(* IEC 61131-3 sources: Simulated-machine/integrations/openplc/thermal-plant-v3, 1 file *)

(* ---- thermal-plant-v3.st ---- *)
(* Generated by tools/generate_openplc_v3_gateway.py.
   OpenPLC Runtime v3 gateway for the self-holding thermal plant.

   The devices start themselves and run their own regulators.  This
   program only exchanges data and evaluates logic; it never computes a
   control value.  The only holding registers written are
   COMMAND_SEQUENCE, WATCHDOG_COUNTER and RESET_KEY.

   Addresses come from the OpenPLC v3 Modbus master image: slave devices
   must be configured in the order listed in slave-devices.csv. *)
PROGRAM main
  VAR
    i_outputs_initialized : BOOL := FALSE;
    i_watchdog_scan_count : UINT := 0;
    i_watchdog_tick : BOOL := FALSE;
    i_plant_comm_lost : BOOL := FALSE;
    i_overspeed : BOOL := FALSE;
    i_overspeed_prev : BOOL := FALSE;
    i_condenser_last_echo : UINT := 0;
    i_condenser_echo_stale_ticks : UINT := 0;
    i_condenser_comm_lost : BOOL := FALSE;
    i_condensate_pump_last_echo : UINT := 0;
    i_condensate_pump_echo_stale_ticks : UINT := 0;
    i_condensate_pump_comm_lost : BOOL := FALSE;
    i_feedwater_tank_last_echo : UINT := 0;
    i_feedwater_tank_echo_stale_ticks : UINT := 0;
    i_feedwater_tank_comm_lost : BOOL := FALSE;
    i_feedwater_pump_last_echo : UINT := 0;
    i_feedwater_pump_echo_stale_ticks : UINT := 0;
    i_feedwater_pump_comm_lost : BOOL := FALSE;
    i_boiler_last_echo : UINT := 0;
    i_boiler_echo_stale_ticks : UINT := 0;
    i_boiler_comm_lost : BOOL := FALSE;
    i_steam_valve_last_echo : UINT := 0;
    i_steam_valve_echo_stale_ticks : UINT := 0;
    i_steam_valve_comm_lost : BOOL := FALSE;
    i_turbine_last_echo : UINT := 0;
    i_turbine_echo_stale_ticks : UINT := 0;
    i_turbine_comm_lost : BOOL := FALSE;
    i_generator_last_echo : UINT := 0;
    i_generator_echo_stale_ticks : UINT := 0;
    i_generator_comm_lost : BOOL := FALSE;
    i_condenser_start_active : BOOL := FALSE;
    i_condenser_start_scans : UINT := 0;
    i_condenser_stop_active : BOOL := FALSE;
    i_condenser_stop_scans : UINT := 0;
    i_condenser_reset_trip_active : BOOL := FALSE;
    i_condenser_reset_trip_scans : UINT := 0;
    i_condenser_ack_alarm_active : BOOL := FALSE;
    i_condenser_ack_alarm_scans : UINT := 0;
    i_condenser_trip_test_active : BOOL := FALSE;
    i_condenser_trip_test_scans : UINT := 0;
    i_condenser_clear_totalizer_active : BOOL := FALSE;
    i_condenser_clear_totalizer_scans : UINT := 0;
    i_condensate_pump_start_active : BOOL := FALSE;
    i_condensate_pump_start_scans : UINT := 0;
    i_condensate_pump_stop_active : BOOL := FALSE;
    i_condensate_pump_stop_scans : UINT := 0;
    i_condensate_pump_reset_trip_active : BOOL := FALSE;
    i_condensate_pump_reset_trip_scans : UINT := 0;
    i_condensate_pump_ack_alarm_active : BOOL := FALSE;
    i_condensate_pump_ack_alarm_scans : UINT := 0;
    i_condensate_pump_trip_test_active : BOOL := FALSE;
    i_condensate_pump_trip_test_scans : UINT := 0;
    i_condensate_pump_clear_totalizer_active : BOOL := FALSE;
    i_condensate_pump_clear_totalizer_scans : UINT := 0;
    i_feedwater_tank_start_active : BOOL := FALSE;
    i_feedwater_tank_start_scans : UINT := 0;
    i_feedwater_tank_stop_active : BOOL := FALSE;
    i_feedwater_tank_stop_scans : UINT := 0;
    i_feedwater_tank_reset_trip_active : BOOL := FALSE;
    i_feedwater_tank_reset_trip_scans : UINT := 0;
    i_feedwater_tank_ack_alarm_active : BOOL := FALSE;
    i_feedwater_tank_ack_alarm_scans : UINT := 0;
    i_feedwater_tank_trip_test_active : BOOL := FALSE;
    i_feedwater_tank_trip_test_scans : UINT := 0;
    i_feedwater_tank_clear_totalizer_active : BOOL := FALSE;
    i_feedwater_tank_clear_totalizer_scans : UINT := 0;
    i_feedwater_pump_start_active : BOOL := FALSE;
    i_feedwater_pump_start_scans : UINT := 0;
    i_feedwater_pump_stop_active : BOOL := FALSE;
    i_feedwater_pump_stop_scans : UINT := 0;
    i_feedwater_pump_reset_trip_active : BOOL := FALSE;
    i_feedwater_pump_reset_trip_scans : UINT := 0;
    i_feedwater_pump_ack_alarm_active : BOOL := FALSE;
    i_feedwater_pump_ack_alarm_scans : UINT := 0;
    i_feedwater_pump_trip_test_active : BOOL := FALSE;
    i_feedwater_pump_trip_test_scans : UINT := 0;
    i_feedwater_pump_clear_totalizer_active : BOOL := FALSE;
    i_feedwater_pump_clear_totalizer_scans : UINT := 0;
    i_boiler_start_active : BOOL := FALSE;
    i_boiler_start_scans : UINT := 0;
    i_boiler_stop_active : BOOL := FALSE;
    i_boiler_stop_scans : UINT := 0;
    i_boiler_reset_trip_active : BOOL := FALSE;
    i_boiler_reset_trip_scans : UINT := 0;
    i_boiler_ack_alarm_active : BOOL := FALSE;
    i_boiler_ack_alarm_scans : UINT := 0;
    i_boiler_trip_test_active : BOOL := FALSE;
    i_boiler_trip_test_scans : UINT := 0;
    i_boiler_clear_totalizer_active : BOOL := FALSE;
    i_boiler_clear_totalizer_scans : UINT := 0;
    i_steam_valve_start_active : BOOL := FALSE;
    i_steam_valve_start_scans : UINT := 0;
    i_steam_valve_stop_active : BOOL := FALSE;
    i_steam_valve_stop_scans : UINT := 0;
    i_steam_valve_reset_trip_active : BOOL := FALSE;
    i_steam_valve_reset_trip_scans : UINT := 0;
    i_steam_valve_ack_alarm_active : BOOL := FALSE;
    i_steam_valve_ack_alarm_scans : UINT := 0;
    i_steam_valve_trip_test_active : BOOL := FALSE;
    i_steam_valve_trip_test_scans : UINT := 0;
    i_steam_valve_clear_totalizer_active : BOOL := FALSE;
    i_steam_valve_clear_totalizer_scans : UINT := 0;
    i_turbine_start_active : BOOL := FALSE;
    i_turbine_start_scans : UINT := 0;
    i_turbine_stop_active : BOOL := FALSE;
    i_turbine_stop_scans : UINT := 0;
    i_turbine_reset_trip_active : BOOL := FALSE;
    i_turbine_reset_trip_scans : UINT := 0;
    i_turbine_ack_alarm_active : BOOL := FALSE;
    i_turbine_ack_alarm_scans : UINT := 0;
    i_turbine_trip_test_active : BOOL := FALSE;
    i_turbine_trip_test_scans : UINT := 0;
    i_turbine_clear_totalizer_active : BOOL := FALSE;
    i_turbine_clear_totalizer_scans : UINT := 0;
    i_generator_start_active : BOOL := FALSE;
    i_generator_start_scans : UINT := 0;
    i_generator_stop_active : BOOL := FALSE;
    i_generator_stop_scans : UINT := 0;
    i_generator_reset_trip_active : BOOL := FALSE;
    i_generator_reset_trip_scans : UINT := 0;
    i_generator_ack_alarm_active : BOOL := FALSE;
    i_generator_ack_alarm_scans : UINT := 0;
    i_generator_trip_test_active : BOOL := FALSE;
    i_generator_trip_test_scans : UINT := 0;
    i_generator_clear_totalizer_active : BOOL := FALSE;
    i_generator_clear_totalizer_scans : UINT := 0;
    i_turbine_trip_prev : BOOL := FALSE;
    i_boiler_trip_prev : BOOL := FALSE;
    i_condenser_trip_prev : BOOL := FALSE;
    i_feedwater_pump_trip_prev : BOOL := FALSE;
    i_condensate_pump_trip_prev : BOOL := FALSE;
    i_steam_valve_trip_prev : BOOL := FALSE;

    condenser__coil__start AT %QX100.0 : BOOL := FALSE;
    condenser__coil__stop AT %QX100.1 : BOOL := FALSE;
    condenser__coil__reset_trip AT %QX100.2 : BOOL := FALSE;
    condenser__coil__ack_alarm AT %QX100.3 : BOOL := FALSE;
    condenser__coil__emergency_stop AT %QX100.4 : BOOL := FALSE;
    condenser__coil__force_safe AT %QX100.5 : BOOL := FALSE;
    condenser__coil__trip_test AT %QX100.6 : BOOL := FALSE;
    condenser__coil__clear_totalizer AT %QX100.7 : BOOL := FALSE;
    condenser__discrete__ready AT %IX100.0 : BOOL := FALSE;
    condenser__discrete__running AT %IX100.1 : BOOL := FALSE;
    condenser__discrete__starting AT %IX100.2 : BOOL := FALSE;
    condenser__discrete__stopping AT %IX100.3 : BOOL := FALSE;
    condenser__discrete__tripped AT %IX100.4 : BOOL := FALSE;
    condenser__discrete__alarm_active AT %IX100.5 : BOOL := FALSE;
    condenser__discrete__local_mode AT %IX100.6 : BOOL := FALSE;
    condenser__discrete__remote_mode AT %IX100.7 : BOOL := FALSE;
    condenser__discrete__auto_mode AT %IX101.0 : BOOL := FALSE;
    condenser__discrete__manual_mode AT %IX101.1 : BOOL := FALSE;
    condenser__discrete__control_watchdog_ok AT %IX101.2 : BOOL := FALSE;
    condenser__discrete__sim_bus_ok AT %IX101.3 : BOOL := FALSE;
    condenser__discrete__interlocks_ok AT %IX101.4 : BOOL := FALSE;
    condenser__discrete__sensor_fault AT %IX101.5 : BOOL := FALSE;
    condenser__discrete__actuator_fault AT %IX101.6 : BOOL := FALSE;
    condenser__discrete__maintenance_mode AT %IX101.7 : BOOL := FALSE;
    condenser__input__status_word AT %IW100 : UINT := 0;
    condenser__input__alarm_word_1 AT %IW101 : UINT := 0;
    condenser__input__alarm_word_2 AT %IW102 : UINT := 0;
    condenser__input__trip_word AT %IW103 : UINT := 0;
    condenser__input__device_state AT %IW104 : UINT := 0;
    condenser__input__first_out_code AT %IW105 : UINT := 0;
    condenser__input__overall_quality AT %IW106 : UINT := 0;
    condenser__input__register_map_version AT %IW107 : UINT := 0;
    condenser__input__firmware_version AT %IW108 : UINT := 0;
    condenser__input__condenser_pressure AT %IW109 : UINT := 0;
    condenser__input__vacuum AT %IW110 : UINT := 0;
    condenser__input__hotwell_level AT %IW111 : UINT := 0;
    condenser__input__exhaust_inflow AT %IW112 : UINT := 0;
    condenser__input__condensing_capacity AT %IW113 : UINT := 0;
    condenser__input__actual_condensed AT %IW114 : UINT := 0;
    condenser__input__condensate_outflow AT %IW115 : UINT := 0;
    condenser__input__cooling_water_availability AT %IW116 : UINT := 0;
    condenser__input__vacuum_system_output AT %IW117 : UINT := 0;
    condenser__input__condensate_temperature AT %IW118 : UINT := 0;
    condenser__input__hotwell_mass_hi AT %IW119 : UINT := 0;
    condenser__input__hotwell_mass_lo AT %IW120 : UINT := 0;
    condenser__input__makeup_valve_position AT %IW121 : UINT := 0;
    condenser__input__makeup_flow AT %IW122 : UINT := 0;
    condenser__input__local_output AT %IW125 : UINT := 0;
    condenser__input__self_hold_state AT %IW126 : UINT := 0;
    condenser__input__permissive_word AT %IW127 : UINT := 0;
    condenser__input__watchdog_echo AT %IW129 : UINT := 0;
    condenser__input__scan_time_ms AT %IW130 : UINT := 0;
    condenser__input__modbus_request_count AT %IW131 : UINT := 0;
    condenser__input__rejected_command_count AT %IW132 : UINT := 0;
    condenser__input__exception_count AT %IW133 : UINT := 0;
    condenser__input__sim_quality_word AT %IW134 : UINT := 0;
    condenser__input__sim_tick_low AT %IW135 : UINT := 0;
    condenser__input__comm_loss_seconds AT %IW136 : UINT := 0;
    condenser__input__fault_inject_word AT %IW137 : UINT := 0;
    condenser__input__snapshot_generation AT %IW138 : UINT := 0;
    condenser__input__run_seconds_hi AT %IW139 : UINT := 0;
    condenser__input__run_seconds_lo AT %IW140 : UINT := 0;
    condenser__input__start_count AT %IW141 : UINT := 0;
    condenser__input__trip_count AT %IW142 : UINT := 0;
    condenser__input__mass_total_hi AT %IW143 : UINT := 0;
    condenser__input__mass_total_lo AT %IW144 : UINT := 0;
    condenser__input__energy_total_hi AT %IW145 : UINT := 0;
    condenser__input__energy_total_lo AT %IW146 : UINT := 0;
    condenser__input__alarm_count AT %IW147 : UINT := 0;
    condenser__input__accepted_command_count AT %IW148 : UINT := 0;
    condenser__holding__command_sequence AT %QW100 : UINT := 0;
    condenser__holding__watchdog_counter AT %QW101 : UINT := 0;
    condenser__holding__reset_key AT %QW102 : UINT := 0;
    condensate_pump__coil__start AT %QX101.0 : BOOL := FALSE;
    condensate_pump__coil__stop AT %QX101.1 : BOOL := FALSE;
    condensate_pump__coil__reset_trip AT %QX101.2 : BOOL := FALSE;
    condensate_pump__coil__ack_alarm AT %QX101.3 : BOOL := FALSE;
    condensate_pump__coil__emergency_stop AT %QX101.4 : BOOL := FALSE;
    condensate_pump__coil__force_safe AT %QX101.5 : BOOL := FALSE;
    condensate_pump__coil__trip_test AT %QX101.6 : BOOL := FALSE;
    condensate_pump__coil__clear_totalizer AT %QX101.7 : BOOL := FALSE;
    condensate_pump__discrete__ready AT %IX102.0 : BOOL := FALSE;
    condensate_pump__discrete__running AT %IX102.1 : BOOL := FALSE;
    condensate_pump__discrete__starting AT %IX102.2 : BOOL := FALSE;
    condensate_pump__discrete__stopping AT %IX102.3 : BOOL := FALSE;
    condensate_pump__discrete__tripped AT %IX102.4 : BOOL := FALSE;
    condensate_pump__discrete__alarm_active AT %IX102.5 : BOOL := FALSE;
    condensate_pump__discrete__local_mode AT %IX102.6 : BOOL := FALSE;
    condensate_pump__discrete__remote_mode AT %IX102.7 : BOOL := FALSE;
    condensate_pump__discrete__auto_mode AT %IX103.0 : BOOL := FALSE;
    condensate_pump__discrete__manual_mode AT %IX103.1 : BOOL := FALSE;
    condensate_pump__discrete__control_watchdog_ok AT %IX103.2 : BOOL := FALSE;
    condensate_pump__discrete__sim_bus_ok AT %IX103.3 : BOOL := FALSE;
    condensate_pump__discrete__interlocks_ok AT %IX103.4 : BOOL := FALSE;
    condensate_pump__discrete__sensor_fault AT %IX103.5 : BOOL := FALSE;
    condensate_pump__discrete__actuator_fault AT %IX103.6 : BOOL := FALSE;
    condensate_pump__discrete__maintenance_mode AT %IX103.7 : BOOL := FALSE;
    condensate_pump__input__status_word AT %IW149 : UINT := 0;
    condensate_pump__input__alarm_word_1 AT %IW150 : UINT := 0;
    condensate_pump__input__alarm_word_2 AT %IW151 : UINT := 0;
    condensate_pump__input__trip_word AT %IW152 : UINT := 0;
    condensate_pump__input__device_state AT %IW153 : UINT := 0;
    condensate_pump__input__first_out_code AT %IW154 : UINT := 0;
    condensate_pump__input__overall_quality AT %IW155 : UINT := 0;
    condensate_pump__input__register_map_version AT %IW156 : UINT := 0;
    condensate_pump__input__firmware_version AT %IW157 : UINT := 0;
    condensate_pump__input__actual_speed AT %IW158 : UINT := 0;
    condensate_pump__input__flow AT %IW159 : UINT := 0;
    condensate_pump__input__suction_pressure AT %IW160 : UINT := 0;
    condensate_pump__input__discharge_pressure AT %IW161 : UINT := 0;
    condensate_pump__input__motor_current AT %IW162 : UINT := 0;
    condensate_pump__input__npsh_margin AT %IW163 : UINT := 0;
    condensate_pump__input__vibration AT %IW164 : UINT := 0;
    condensate_pump__input__source_level AT %IW165 : UINT := 0;
    condensate_pump__input__backpressure AT %IW166 : UINT := 0;
    condensate_pump__input__outlet_valve_position AT %IW167 : UINT := 0;
    condensate_pump__input__cavitation_factor AT %IW168 : UINT := 0;
    condensate_pump__input__local_output AT %IW174 : UINT := 0;
    condensate_pump__input__self_hold_state AT %IW175 : UINT := 0;
    condensate_pump__input__permissive_word AT %IW176 : UINT := 0;
    condensate_pump__input__watchdog_echo AT %IW178 : UINT := 0;
    condensate_pump__input__scan_time_ms AT %IW179 : UINT := 0;
    condensate_pump__input__modbus_request_count AT %IW180 : UINT := 0;
    condensate_pump__input__rejected_command_count AT %IW181 : UINT := 0;
    condensate_pump__input__exception_count AT %IW182 : UINT := 0;
    condensate_pump__input__sim_quality_word AT %IW183 : UINT := 0;
    condensate_pump__input__sim_tick_low AT %IW184 : UINT := 0;
    condensate_pump__input__comm_loss_seconds AT %IW185 : UINT := 0;
    condensate_pump__input__fault_inject_word AT %IW186 : UINT := 0;
    condensate_pump__input__snapshot_generation AT %IW187 : UINT := 0;
    condensate_pump__input__run_seconds_hi AT %IW188 : UINT := 0;
    condensate_pump__input__run_seconds_lo AT %IW189 : UINT := 0;
    condensate_pump__input__start_count AT %IW190 : UINT := 0;
    condensate_pump__input__trip_count AT %IW191 : UINT := 0;
    condensate_pump__input__mass_total_hi AT %IW192 : UINT := 0;
    condensate_pump__input__mass_total_lo AT %IW193 : UINT := 0;
    condensate_pump__input__energy_total_hi AT %IW194 : UINT := 0;
    condensate_pump__input__energy_total_lo AT %IW195 : UINT := 0;
    condensate_pump__input__alarm_count AT %IW196 : UINT := 0;
    condensate_pump__input__accepted_command_count AT %IW197 : UINT := 0;
    condensate_pump__holding__command_sequence AT %QW103 : UINT := 0;
    condensate_pump__holding__watchdog_counter AT %QW104 : UINT := 0;
    condensate_pump__holding__reset_key AT %QW105 : UINT := 0;
    feedwater_tank__coil__start AT %QX102.0 : BOOL := FALSE;
    feedwater_tank__coil__stop AT %QX102.1 : BOOL := FALSE;
    feedwater_tank__coil__reset_trip AT %QX102.2 : BOOL := FALSE;
    feedwater_tank__coil__ack_alarm AT %QX102.3 : BOOL := FALSE;
    feedwater_tank__coil__emergency_stop AT %QX102.4 : BOOL := FALSE;
    feedwater_tank__coil__force_safe AT %QX102.5 : BOOL := FALSE;
    feedwater_tank__coil__trip_test AT %QX102.6 : BOOL := FALSE;
    feedwater_tank__coil__clear_totalizer AT %QX102.7 : BOOL := FALSE;
    feedwater_tank__discrete__ready AT %IX104.0 : BOOL := FALSE;
    feedwater_tank__discrete__running AT %IX104.1 : BOOL := FALSE;
    feedwater_tank__discrete__starting AT %IX104.2 : BOOL := FALSE;
    feedwater_tank__discrete__stopping AT %IX104.3 : BOOL := FALSE;
    feedwater_tank__discrete__tripped AT %IX104.4 : BOOL := FALSE;
    feedwater_tank__discrete__alarm_active AT %IX104.5 : BOOL := FALSE;
    feedwater_tank__discrete__local_mode AT %IX104.6 : BOOL := FALSE;
    feedwater_tank__discrete__remote_mode AT %IX104.7 : BOOL := FALSE;
    feedwater_tank__discrete__auto_mode AT %IX105.0 : BOOL := FALSE;
    feedwater_tank__discrete__manual_mode AT %IX105.1 : BOOL := FALSE;
    feedwater_tank__discrete__control_watchdog_ok AT %IX105.2 : BOOL := FALSE;
    feedwater_tank__discrete__sim_bus_ok AT %IX105.3 : BOOL := FALSE;
    feedwater_tank__discrete__interlocks_ok AT %IX105.4 : BOOL := FALSE;
    feedwater_tank__discrete__sensor_fault AT %IX105.5 : BOOL := FALSE;
    feedwater_tank__discrete__actuator_fault AT %IX105.6 : BOOL := FALSE;
    feedwater_tank__discrete__maintenance_mode AT %IX105.7 : BOOL := FALSE;
    feedwater_tank__input__status_word AT %IW198 : UINT := 0;
    feedwater_tank__input__alarm_word_1 AT %IW199 : UINT := 0;
    feedwater_tank__input__alarm_word_2 AT %IW200 : UINT := 0;
    feedwater_tank__input__trip_word AT %IW201 : UINT := 0;
    feedwater_tank__input__device_state AT %IW202 : UINT := 0;
    feedwater_tank__input__first_out_code AT %IW203 : UINT := 0;
    feedwater_tank__input__overall_quality AT %IW204 : UINT := 0;
    feedwater_tank__input__register_map_version AT %IW205 : UINT := 0;
    feedwater_tank__input__firmware_version AT %IW206 : UINT := 0;
    feedwater_tank__input__tank_level AT %IW207 : UINT := 0;
    feedwater_tank__input__tank_mass_hi AT %IW208 : UINT := 0;
    feedwater_tank__input__tank_mass_lo AT %IW209 : UINT := 0;
    feedwater_tank__input__condensate_inflow AT %IW210 : UINT := 0;
    feedwater_tank__input__feedwater_outflow AT %IW211 : UINT := 0;
    feedwater_tank__input__water_temperature AT %IW212 : UINT := 0;
    feedwater_tank__input__tank_pressure AT %IW213 : UINT := 0;
    feedwater_tank__input__overflow_flow AT %IW214 : UINT := 0;
    feedwater_tank__input__net_flow AT %IW215 : UINT := 0;
    feedwater_tank__input__local_output AT %IW223 : UINT := 0;
    feedwater_tank__input__self_hold_state AT %IW224 : UINT := 0;
    feedwater_tank__input__permissive_word AT %IW225 : UINT := 0;
    feedwater_tank__input__watchdog_echo AT %IW227 : UINT := 0;
    feedwater_tank__input__scan_time_ms AT %IW228 : UINT := 0;
    feedwater_tank__input__modbus_request_count AT %IW229 : UINT := 0;
    feedwater_tank__input__rejected_command_count AT %IW230 : UINT := 0;
    feedwater_tank__input__exception_count AT %IW231 : UINT := 0;
    feedwater_tank__input__sim_quality_word AT %IW232 : UINT := 0;
    feedwater_tank__input__sim_tick_low AT %IW233 : UINT := 0;
    feedwater_tank__input__comm_loss_seconds AT %IW234 : UINT := 0;
    feedwater_tank__input__fault_inject_word AT %IW235 : UINT := 0;
    feedwater_tank__input__snapshot_generation AT %IW236 : UINT := 0;
    feedwater_tank__input__run_seconds_hi AT %IW237 : UINT := 0;
    feedwater_tank__input__run_seconds_lo AT %IW238 : UINT := 0;
    feedwater_tank__input__start_count AT %IW239 : UINT := 0;
    feedwater_tank__input__trip_count AT %IW240 : UINT := 0;
    feedwater_tank__input__mass_total_hi AT %IW241 : UINT := 0;
    feedwater_tank__input__mass_total_lo AT %IW242 : UINT := 0;
    feedwater_tank__input__energy_total_hi AT %IW243 : UINT := 0;
    feedwater_tank__input__energy_total_lo AT %IW244 : UINT := 0;
    feedwater_tank__input__alarm_count AT %IW245 : UINT := 0;
    feedwater_tank__input__accepted_command_count AT %IW246 : UINT := 0;
    feedwater_tank__holding__command_sequence AT %QW106 : UINT := 0;
    feedwater_tank__holding__watchdog_counter AT %QW107 : UINT := 0;
    feedwater_tank__holding__reset_key AT %QW108 : UINT := 0;
    feedwater_pump__coil__start AT %QX103.0 : BOOL := FALSE;
    feedwater_pump__coil__stop AT %QX103.1 : BOOL := FALSE;
    feedwater_pump__coil__reset_trip AT %QX103.2 : BOOL := FALSE;
    feedwater_pump__coil__ack_alarm AT %QX103.3 : BOOL := FALSE;
    feedwater_pump__coil__emergency_stop AT %QX103.4 : BOOL := FALSE;
    feedwater_pump__coil__force_safe AT %QX103.5 : BOOL := FALSE;
    feedwater_pump__coil__trip_test AT %QX103.6 : BOOL := FALSE;
    feedwater_pump__coil__clear_totalizer AT %QX103.7 : BOOL := FALSE;
    feedwater_pump__discrete__ready AT %IX106.0 : BOOL := FALSE;
    feedwater_pump__discrete__running AT %IX106.1 : BOOL := FALSE;
    feedwater_pump__discrete__starting AT %IX106.2 : BOOL := FALSE;
    feedwater_pump__discrete__stopping AT %IX106.3 : BOOL := FALSE;
    feedwater_pump__discrete__tripped AT %IX106.4 : BOOL := FALSE;
    feedwater_pump__discrete__alarm_active AT %IX106.5 : BOOL := FALSE;
    feedwater_pump__discrete__local_mode AT %IX106.6 : BOOL := FALSE;
    feedwater_pump__discrete__remote_mode AT %IX106.7 : BOOL := FALSE;
    feedwater_pump__discrete__auto_mode AT %IX107.0 : BOOL := FALSE;
    feedwater_pump__discrete__manual_mode AT %IX107.1 : BOOL := FALSE;
    feedwater_pump__discrete__control_watchdog_ok AT %IX107.2 : BOOL := FALSE;
    feedwater_pump__discrete__sim_bus_ok AT %IX107.3 : BOOL := FALSE;
    feedwater_pump__discrete__interlocks_ok AT %IX107.4 : BOOL := FALSE;
    feedwater_pump__discrete__sensor_fault AT %IX107.5 : BOOL := FALSE;
    feedwater_pump__discrete__actuator_fault AT %IX107.6 : BOOL := FALSE;
    feedwater_pump__discrete__maintenance_mode AT %IX107.7 : BOOL := FALSE;
    feedwater_pump__input__status_word AT %IW247 : UINT := 0;
    feedwater_pump__input__alarm_word_1 AT %IW248 : UINT := 0;
    feedwater_pump__input__alarm_word_2 AT %IW249 : UINT := 0;
    feedwater_pump__input__trip_word AT %IW250 : UINT := 0;
    feedwater_pump__input__device_state AT %IW251 : UINT := 0;
    feedwater_pump__input__first_out_code AT %IW252 : UINT := 0;
    feedwater_pump__input__overall_quality AT %IW253 : UINT := 0;
    feedwater_pump__input__register_map_version AT %IW254 : UINT := 0;
    feedwater_pump__input__firmware_version AT %IW255 : UINT := 0;
    feedwater_pump__input__actual_speed AT %IW256 : UINT := 0;
    feedwater_pump__input__flow AT %IW257 : UINT := 0;
    feedwater_pump__input__suction_pressure AT %IW258 : UINT := 0;
    feedwater_pump__input__discharge_pressure AT %IW259 : UINT := 0;
    feedwater_pump__input__motor_current AT %IW260 : UINT := 0;
    feedwater_pump__input__npsh_margin AT %IW261 : UINT := 0;
    feedwater_pump__input__vibration AT %IW262 : UINT := 0;
    feedwater_pump__input__source_level AT %IW263 : UINT := 0;
    feedwater_pump__input__backpressure AT %IW264 : UINT := 0;
    feedwater_pump__input__outlet_valve_position AT %IW265 : UINT := 0;
    feedwater_pump__input__cavitation_factor AT %IW266 : UINT := 0;
    feedwater_pump__input__boiler_pressure AT %IW267 : UINT := 0;
    feedwater_pump__input__feedwater_permitted AT %IW268 : UINT := 0;
    feedwater_pump__input__local_output AT %IW272 : UINT := 0;
    feedwater_pump__input__self_hold_state AT %IW273 : UINT := 0;
    feedwater_pump__input__permissive_word AT %IW274 : UINT := 0;
    feedwater_pump__input__watchdog_echo AT %IW276 : UINT := 0;
    feedwater_pump__input__scan_time_ms AT %IW277 : UINT := 0;
    feedwater_pump__input__modbus_request_count AT %IW278 : UINT := 0;
    feedwater_pump__input__rejected_command_count AT %IW279 : UINT := 0;
    feedwater_pump__input__exception_count AT %IW280 : UINT := 0;
    feedwater_pump__input__sim_quality_word AT %IW281 : UINT := 0;
    feedwater_pump__input__sim_tick_low AT %IW282 : UINT := 0;
    feedwater_pump__input__comm_loss_seconds AT %IW283 : UINT := 0;
    feedwater_pump__input__fault_inject_word AT %IW284 : UINT := 0;
    feedwater_pump__input__snapshot_generation AT %IW285 : UINT := 0;
    feedwater_pump__input__run_seconds_hi AT %IW286 : UINT := 0;
    feedwater_pump__input__run_seconds_lo AT %IW287 : UINT := 0;
    feedwater_pump__input__start_count AT %IW288 : UINT := 0;
    feedwater_pump__input__trip_count AT %IW289 : UINT := 0;
    feedwater_pump__input__mass_total_hi AT %IW290 : UINT := 0;
    feedwater_pump__input__mass_total_lo AT %IW291 : UINT := 0;
    feedwater_pump__input__energy_total_hi AT %IW292 : UINT := 0;
    feedwater_pump__input__energy_total_lo AT %IW293 : UINT := 0;
    feedwater_pump__input__alarm_count AT %IW294 : UINT := 0;
    feedwater_pump__input__accepted_command_count AT %IW295 : UINT := 0;
    feedwater_pump__holding__command_sequence AT %QW109 : UINT := 0;
    feedwater_pump__holding__watchdog_counter AT %QW110 : UINT := 0;
    feedwater_pump__holding__reset_key AT %QW111 : UINT := 0;
    boiler__coil__start AT %QX104.0 : BOOL := FALSE;
    boiler__coil__stop AT %QX104.1 : BOOL := FALSE;
    boiler__coil__reset_trip AT %QX104.2 : BOOL := FALSE;
    boiler__coil__ack_alarm AT %QX104.3 : BOOL := FALSE;
    boiler__coil__emergency_stop AT %QX104.4 : BOOL := FALSE;
    boiler__coil__force_safe AT %QX104.5 : BOOL := FALSE;
    boiler__coil__trip_test AT %QX104.6 : BOOL := FALSE;
    boiler__coil__clear_totalizer AT %QX104.7 : BOOL := FALSE;
    boiler__discrete__ready AT %IX108.0 : BOOL := FALSE;
    boiler__discrete__running AT %IX108.1 : BOOL := FALSE;
    boiler__discrete__starting AT %IX108.2 : BOOL := FALSE;
    boiler__discrete__stopping AT %IX108.3 : BOOL := FALSE;
    boiler__discrete__tripped AT %IX108.4 : BOOL := FALSE;
    boiler__discrete__alarm_active AT %IX108.5 : BOOL := FALSE;
    boiler__discrete__local_mode AT %IX108.6 : BOOL := FALSE;
    boiler__discrete__remote_mode AT %IX108.7 : BOOL := FALSE;
    boiler__discrete__auto_mode AT %IX109.0 : BOOL := FALSE;
    boiler__discrete__manual_mode AT %IX109.1 : BOOL := FALSE;
    boiler__discrete__control_watchdog_ok AT %IX109.2 : BOOL := FALSE;
    boiler__discrete__sim_bus_ok AT %IX109.3 : BOOL := FALSE;
    boiler__discrete__interlocks_ok AT %IX109.4 : BOOL := FALSE;
    boiler__discrete__sensor_fault AT %IX109.5 : BOOL := FALSE;
    boiler__discrete__actuator_fault AT %IX109.6 : BOOL := FALSE;
    boiler__discrete__maintenance_mode AT %IX109.7 : BOOL := FALSE;
    boiler__input__status_word AT %IW296 : UINT := 0;
    boiler__input__alarm_word_1 AT %IW297 : UINT := 0;
    boiler__input__alarm_word_2 AT %IW298 : UINT := 0;
    boiler__input__trip_word AT %IW299 : UINT := 0;
    boiler__input__device_state AT %IW300 : UINT := 0;
    boiler__input__first_out_code AT %IW301 : UINT := 0;
    boiler__input__overall_quality AT %IW302 : UINT := 0;
    boiler__input__register_map_version AT %IW303 : UINT := 0;
    boiler__input__firmware_version AT %IW304 : UINT := 0;
    boiler__input__boiler_pressure AT %IW305 : UINT := 0;
    boiler__input__level_indicated AT %IW306 : UINT := 0;
    boiler__input__level_actual AT %IW307 : UINT := 0;
    boiler__input__feedwater_flow AT %IW308 : UINT := 0;
    boiler__input__steam_generation AT %IW309 : UINT := 0;
    boiler__input__steam_outflow AT %IW310 : UINT := 0;
    boiler__input__burner_output AT %IW311 : UINT := 0;
    boiler__input__steam_temperature AT %IW312 : UINT := 0;
    boiler__input__water_mass_hi AT %IW313 : UINT := 0;
    boiler__input__water_mass_lo AT %IW314 : UINT := 0;
    boiler__input__flame_status AT %IW315 : UINT := 0;
    boiler__input__blowdown_flow AT %IW316 : UINT := 0;
    boiler__input__purge_time_remaining AT %IW317 : UINT := 0;
    boiler__input__feedwater_permitted AT %IW318 : UINT := 0;
    boiler__input__relief_flow AT %IW319 : UINT := 0;
    boiler__input__local_output AT %IW321 : UINT := 0;
    boiler__input__self_hold_state AT %IW322 : UINT := 0;
    boiler__input__permissive_word AT %IW323 : UINT := 0;
    boiler__input__watchdog_echo AT %IW325 : UINT := 0;
    boiler__input__scan_time_ms AT %IW326 : UINT := 0;
    boiler__input__modbus_request_count AT %IW327 : UINT := 0;
    boiler__input__rejected_command_count AT %IW328 : UINT := 0;
    boiler__input__exception_count AT %IW329 : UINT := 0;
    boiler__input__sim_quality_word AT %IW330 : UINT := 0;
    boiler__input__sim_tick_low AT %IW331 : UINT := 0;
    boiler__input__comm_loss_seconds AT %IW332 : UINT := 0;
    boiler__input__fault_inject_word AT %IW333 : UINT := 0;
    boiler__input__snapshot_generation AT %IW334 : UINT := 0;
    boiler__input__run_seconds_hi AT %IW335 : UINT := 0;
    boiler__input__run_seconds_lo AT %IW336 : UINT := 0;
    boiler__input__start_count AT %IW337 : UINT := 0;
    boiler__input__trip_count AT %IW338 : UINT := 0;
    boiler__input__mass_total_hi AT %IW339 : UINT := 0;
    boiler__input__mass_total_lo AT %IW340 : UINT := 0;
    boiler__input__energy_total_hi AT %IW341 : UINT := 0;
    boiler__input__energy_total_lo AT %IW342 : UINT := 0;
    boiler__input__alarm_count AT %IW343 : UINT := 0;
    boiler__input__accepted_command_count AT %IW344 : UINT := 0;
    boiler__holding__command_sequence AT %QW112 : UINT := 0;
    boiler__holding__watchdog_counter AT %QW113 : UINT := 0;
    boiler__holding__reset_key AT %QW114 : UINT := 0;
    steam_valve__coil__start AT %QX105.0 : BOOL := FALSE;
    steam_valve__coil__stop AT %QX105.1 : BOOL := FALSE;
    steam_valve__coil__reset_trip AT %QX105.2 : BOOL := FALSE;
    steam_valve__coil__ack_alarm AT %QX105.3 : BOOL := FALSE;
    steam_valve__coil__emergency_stop AT %QX105.4 : BOOL := FALSE;
    steam_valve__coil__force_safe AT %QX105.5 : BOOL := FALSE;
    steam_valve__coil__trip_test AT %QX105.6 : BOOL := FALSE;
    steam_valve__coil__clear_totalizer AT %QX105.7 : BOOL := FALSE;
    steam_valve__discrete__ready AT %IX110.0 : BOOL := FALSE;
    steam_valve__discrete__running AT %IX110.1 : BOOL := FALSE;
    steam_valve__discrete__starting AT %IX110.2 : BOOL := FALSE;
    steam_valve__discrete__stopping AT %IX110.3 : BOOL := FALSE;
    steam_valve__discrete__tripped AT %IX110.4 : BOOL := FALSE;
    steam_valve__discrete__alarm_active AT %IX110.5 : BOOL := FALSE;
    steam_valve__discrete__local_mode AT %IX110.6 : BOOL := FALSE;
    steam_valve__discrete__remote_mode AT %IX110.7 : BOOL := FALSE;
    steam_valve__discrete__auto_mode AT %IX111.0 : BOOL := FALSE;
    steam_valve__discrete__manual_mode AT %IX111.1 : BOOL := FALSE;
    steam_valve__discrete__control_watchdog_ok AT %IX111.2 : BOOL := FALSE;
    steam_valve__discrete__sim_bus_ok AT %IX111.3 : BOOL := FALSE;
    steam_valve__discrete__interlocks_ok AT %IX111.4 : BOOL := FALSE;
    steam_valve__discrete__sensor_fault AT %IX111.5 : BOOL := FALSE;
    steam_valve__discrete__actuator_fault AT %IX111.6 : BOOL := FALSE;
    steam_valve__discrete__maintenance_mode AT %IX111.7 : BOOL := FALSE;
    steam_valve__input__status_word AT %IW345 : UINT := 0;
    steam_valve__input__alarm_word_1 AT %IW346 : UINT := 0;
    steam_valve__input__alarm_word_2 AT %IW347 : UINT := 0;
    steam_valve__input__trip_word AT %IW348 : UINT := 0;
    steam_valve__input__device_state AT %IW349 : UINT := 0;
    steam_valve__input__first_out_code AT %IW350 : UINT := 0;
    steam_valve__input__overall_quality AT %IW351 : UINT := 0;
    steam_valve__input__register_map_version AT %IW352 : UINT := 0;
    steam_valve__input__firmware_version AT %IW353 : UINT := 0;
    steam_valve__input__command_position AT %IW354 : UINT := 0;
    steam_valve__input__actual_position AT %IW355 : UINT := 0;
    steam_valve__input__upstream_pressure AT %IW356 : UINT := 0;
    steam_valve__input__downstream_pressure AT %IW357 : UINT := 0;
    steam_valve__input__steam_flow AT %IW358 : UINT := 0;
    steam_valve__input__steam_temperature AT %IW359 : UINT := 0;
    steam_valve__input__actuator_speed AT %IW360 : UINT := 0;
    steam_valve__input__position_deviation AT %IW361 : UINT := 0;
    steam_valve__input__fast_close_status AT %IW362 : UINT := 0;
    steam_valve__input__valve_fault_code AT %IW363 : UINT := 0;
    steam_valve__input__local_output AT %IW370 : UINT := 0;
    steam_valve__input__self_hold_state AT %IW371 : UINT := 0;
    steam_valve__input__permissive_word AT %IW372 : UINT := 0;
    steam_valve__input__watchdog_echo AT %IW374 : UINT := 0;
    steam_valve__input__scan_time_ms AT %IW375 : UINT := 0;
    steam_valve__input__modbus_request_count AT %IW376 : UINT := 0;
    steam_valve__input__rejected_command_count AT %IW377 : UINT := 0;
    steam_valve__input__exception_count AT %IW378 : UINT := 0;
    steam_valve__input__sim_quality_word AT %IW379 : UINT := 0;
    steam_valve__input__sim_tick_low AT %IW380 : UINT := 0;
    steam_valve__input__comm_loss_seconds AT %IW381 : UINT := 0;
    steam_valve__input__fault_inject_word AT %IW382 : UINT := 0;
    steam_valve__input__snapshot_generation AT %IW383 : UINT := 0;
    steam_valve__input__run_seconds_hi AT %IW384 : UINT := 0;
    steam_valve__input__run_seconds_lo AT %IW385 : UINT := 0;
    steam_valve__input__start_count AT %IW386 : UINT := 0;
    steam_valve__input__trip_count AT %IW387 : UINT := 0;
    steam_valve__input__mass_total_hi AT %IW388 : UINT := 0;
    steam_valve__input__mass_total_lo AT %IW389 : UINT := 0;
    steam_valve__input__energy_total_hi AT %IW390 : UINT := 0;
    steam_valve__input__energy_total_lo AT %IW391 : UINT := 0;
    steam_valve__input__alarm_count AT %IW392 : UINT := 0;
    steam_valve__input__accepted_command_count AT %IW393 : UINT := 0;
    steam_valve__holding__command_sequence AT %QW115 : UINT := 0;
    steam_valve__holding__watchdog_counter AT %QW116 : UINT := 0;
    steam_valve__holding__reset_key AT %QW117 : UINT := 0;
    turbine__coil__start AT %QX106.0 : BOOL := FALSE;
    turbine__coil__stop AT %QX106.1 : BOOL := FALSE;
    turbine__coil__reset_trip AT %QX106.2 : BOOL := FALSE;
    turbine__coil__ack_alarm AT %QX106.3 : BOOL := FALSE;
    turbine__coil__emergency_stop AT %QX106.4 : BOOL := FALSE;
    turbine__coil__force_safe AT %QX106.5 : BOOL := FALSE;
    turbine__coil__trip_test AT %QX106.6 : BOOL := FALSE;
    turbine__coil__clear_totalizer AT %QX106.7 : BOOL := FALSE;
    turbine__discrete__ready AT %IX112.0 : BOOL := FALSE;
    turbine__discrete__running AT %IX112.1 : BOOL := FALSE;
    turbine__discrete__starting AT %IX112.2 : BOOL := FALSE;
    turbine__discrete__stopping AT %IX112.3 : BOOL := FALSE;
    turbine__discrete__tripped AT %IX112.4 : BOOL := FALSE;
    turbine__discrete__alarm_active AT %IX112.5 : BOOL := FALSE;
    turbine__discrete__local_mode AT %IX112.6 : BOOL := FALSE;
    turbine__discrete__remote_mode AT %IX112.7 : BOOL := FALSE;
    turbine__discrete__auto_mode AT %IX113.0 : BOOL := FALSE;
    turbine__discrete__manual_mode AT %IX113.1 : BOOL := FALSE;
    turbine__discrete__control_watchdog_ok AT %IX113.2 : BOOL := FALSE;
    turbine__discrete__sim_bus_ok AT %IX113.3 : BOOL := FALSE;
    turbine__discrete__interlocks_ok AT %IX113.4 : BOOL := FALSE;
    turbine__discrete__sensor_fault AT %IX113.5 : BOOL := FALSE;
    turbine__discrete__actuator_fault AT %IX113.6 : BOOL := FALSE;
    turbine__discrete__maintenance_mode AT %IX113.7 : BOOL := FALSE;
    turbine__input__status_word AT %IW394 : UINT := 0;
    turbine__input__alarm_word_1 AT %IW395 : UINT := 0;
    turbine__input__alarm_word_2 AT %IW396 : UINT := 0;
    turbine__input__trip_word AT %IW397 : UINT := 0;
    turbine__input__device_state AT %IW398 : UINT := 0;
    turbine__input__first_out_code AT %IW399 : UINT := 0;
    turbine__input__overall_quality AT %IW400 : UINT := 0;
    turbine__input__register_map_version AT %IW401 : UINT := 0;
    turbine__input__firmware_version AT %IW402 : UINT := 0;
    turbine__input__speed_rpm AT %IW403 : UINT := 0;
    turbine__input__mechanical_power AT %IW404 : UINT := 0;
    turbine__input__steam_flow AT %IW405 : UINT := 0;
    turbine__input__exhaust_flow AT %IW406 : UINT := 0;
    turbine__input__main_steam_pressure AT %IW407 : UINT := 0;
    turbine__input__exhaust_pressure AT %IW408 : UINT := 0;
    turbine__input__vibration AT %IW409 : UINT := 0;
    turbine__input__bearing_temperature AT %IW410 : UINT := 0;
    turbine__input__governor_output AT %IW411 : UINT := 0;
    turbine__input__acceleration AT %IW412 : UINT := 0;
    turbine__input__efficiency AT %IW413 : UINT := 0;
    turbine__input__local_output AT %IW419 : UINT := 0;
    turbine__input__self_hold_state AT %IW420 : UINT := 0;
    turbine__input__permissive_word AT %IW421 : UINT := 0;
    turbine__input__watchdog_echo AT %IW423 : UINT := 0;
    turbine__input__scan_time_ms AT %IW424 : UINT := 0;
    turbine__input__modbus_request_count AT %IW425 : UINT := 0;
    turbine__input__rejected_command_count AT %IW426 : UINT := 0;
    turbine__input__exception_count AT %IW427 : UINT := 0;
    turbine__input__sim_quality_word AT %IW428 : UINT := 0;
    turbine__input__sim_tick_low AT %IW429 : UINT := 0;
    turbine__input__comm_loss_seconds AT %IW430 : UINT := 0;
    turbine__input__fault_inject_word AT %IW431 : UINT := 0;
    turbine__input__snapshot_generation AT %IW432 : UINT := 0;
    turbine__input__run_seconds_hi AT %IW433 : UINT := 0;
    turbine__input__run_seconds_lo AT %IW434 : UINT := 0;
    turbine__input__start_count AT %IW435 : UINT := 0;
    turbine__input__trip_count AT %IW436 : UINT := 0;
    turbine__input__mass_total_hi AT %IW437 : UINT := 0;
    turbine__input__mass_total_lo AT %IW438 : UINT := 0;
    turbine__input__energy_total_hi AT %IW439 : UINT := 0;
    turbine__input__energy_total_lo AT %IW440 : UINT := 0;
    turbine__input__alarm_count AT %IW441 : UINT := 0;
    turbine__input__accepted_command_count AT %IW442 : UINT := 0;
    turbine__holding__command_sequence AT %QW118 : UINT := 0;
    turbine__holding__watchdog_counter AT %QW119 : UINT := 0;
    turbine__holding__reset_key AT %QW120 : UINT := 0;
    generator__coil__start AT %QX107.0 : BOOL := FALSE;
    generator__coil__stop AT %QX107.1 : BOOL := FALSE;
    generator__coil__reset_trip AT %QX107.2 : BOOL := FALSE;
    generator__coil__ack_alarm AT %QX107.3 : BOOL := FALSE;
    generator__coil__emergency_stop AT %QX107.4 : BOOL := FALSE;
    generator__coil__force_safe AT %QX107.5 : BOOL := FALSE;
    generator__coil__trip_test AT %QX107.6 : BOOL := FALSE;
    generator__coil__clear_totalizer AT %QX107.7 : BOOL := FALSE;
    generator__discrete__ready AT %IX114.0 : BOOL := FALSE;
    generator__discrete__running AT %IX114.1 : BOOL := FALSE;
    generator__discrete__starting AT %IX114.2 : BOOL := FALSE;
    generator__discrete__stopping AT %IX114.3 : BOOL := FALSE;
    generator__discrete__tripped AT %IX114.4 : BOOL := FALSE;
    generator__discrete__alarm_active AT %IX114.5 : BOOL := FALSE;
    generator__discrete__local_mode AT %IX114.6 : BOOL := FALSE;
    generator__discrete__remote_mode AT %IX114.7 : BOOL := FALSE;
    generator__discrete__auto_mode AT %IX115.0 : BOOL := FALSE;
    generator__discrete__manual_mode AT %IX115.1 : BOOL := FALSE;
    generator__discrete__control_watchdog_ok AT %IX115.2 : BOOL := FALSE;
    generator__discrete__sim_bus_ok AT %IX115.3 : BOOL := FALSE;
    generator__discrete__interlocks_ok AT %IX115.4 : BOOL := FALSE;
    generator__discrete__sensor_fault AT %IX115.5 : BOOL := FALSE;
    generator__discrete__actuator_fault AT %IX115.6 : BOOL := FALSE;
    generator__discrete__maintenance_mode AT %IX115.7 : BOOL := FALSE;
    generator__input__status_word AT %IW443 : UINT := 0;
    generator__input__alarm_word_1 AT %IW444 : UINT := 0;
    generator__input__alarm_word_2 AT %IW445 : UINT := 0;
    generator__input__trip_word AT %IW446 : UINT := 0;
    generator__input__device_state AT %IW447 : UINT := 0;
    generator__input__first_out_code AT %IW448 : UINT := 0;
    generator__input__overall_quality AT %IW449 : UINT := 0;
    generator__input__register_map_version AT %IW450 : UINT := 0;
    generator__input__firmware_version AT %IW451 : UINT := 0;
    generator__input__electrical_power AT %IW452 : UINT := 0;
    generator__input__load_demand AT %IW453 : UINT := 0;
    generator__input__frequency AT %IW454 : UINT := 0;
    generator__input__voltage AT %IW455 : UINT := 0;
    generator__input__current AT %IW456 : UINT := 0;
    generator__input__power_factor AT %IW457 : UINT := 0;
    generator__input__breaker_status AT %IW458 : UINT := 0;
    generator__input__sync_permissive AT %IW459 : UINT := 0;
    generator__input__phase_angle_diff AT %IW460 : UINT := 0;
    generator__input__electrical_torque AT %IW461 : UINT := 0;
    generator__input__operating_mode AT %IW462 : UINT := 0;
    generator__input__local_output AT %IW468 : UINT := 0;
    generator__input__self_hold_state AT %IW469 : UINT := 0;
    generator__input__permissive_word AT %IW470 : UINT := 0;
    generator__input__watchdog_echo AT %IW472 : UINT := 0;
    generator__input__scan_time_ms AT %IW473 : UINT := 0;
    generator__input__modbus_request_count AT %IW474 : UINT := 0;
    generator__input__rejected_command_count AT %IW475 : UINT := 0;
    generator__input__exception_count AT %IW476 : UINT := 0;
    generator__input__sim_quality_word AT %IW477 : UINT := 0;
    generator__input__sim_tick_low AT %IW478 : UINT := 0;
    generator__input__comm_loss_seconds AT %IW479 : UINT := 0;
    generator__input__fault_inject_word AT %IW480 : UINT := 0;
    generator__input__snapshot_generation AT %IW481 : UINT := 0;
    generator__input__run_seconds_hi AT %IW482 : UINT := 0;
    generator__input__run_seconds_lo AT %IW483 : UINT := 0;
    generator__input__start_count AT %IW484 : UINT := 0;
    generator__input__trip_count AT %IW485 : UINT := 0;
    generator__input__mass_total_hi AT %IW486 : UINT := 0;
    generator__input__mass_total_lo AT %IW487 : UINT := 0;
    generator__input__energy_total_hi AT %IW488 : UINT := 0;
    generator__input__energy_total_lo AT %IW489 : UINT := 0;
    generator__input__alarm_count AT %IW490 : UINT := 0;
    generator__input__accepted_command_count AT %IW491 : UINT := 0;
    generator__holding__command_sequence AT %QW121 : UINT := 0;
    generator__holding__watchdog_counter AT %QW122 : UINT := 0;
    generator__holding__reset_key AT %QW123 : UINT := 0;
  END_VAR

  (* First scan: arm the watchdogs.  Nothing else is ever written. *)
  IF NOT i_outputs_initialized THEN
    condenser__holding__watchdog_counter := 1;
    condenser__holding__command_sequence := 0;
    condenser__holding__reset_key := 0;
    condensate_pump__holding__watchdog_counter := 1;
    condensate_pump__holding__command_sequence := 0;
    condensate_pump__holding__reset_key := 0;
    feedwater_tank__holding__watchdog_counter := 1;
    feedwater_tank__holding__command_sequence := 0;
    feedwater_tank__holding__reset_key := 0;
    feedwater_pump__holding__watchdog_counter := 1;
    feedwater_pump__holding__command_sequence := 0;
    feedwater_pump__holding__reset_key := 0;
    boiler__holding__watchdog_counter := 1;
    boiler__holding__command_sequence := 0;
    boiler__holding__reset_key := 0;
    steam_valve__holding__watchdog_counter := 1;
    steam_valve__holding__command_sequence := 0;
    steam_valve__holding__reset_key := 0;
    turbine__holding__watchdog_counter := 1;
    turbine__holding__command_sequence := 0;
    turbine__holding__reset_key := 0;
    generator__holding__watchdog_counter := 1;
    generator__holding__command_sequence := 0;
    generator__holding__reset_key := 0;
    i_outputs_initialized := TRUE;
  END_IF;

  (* 200 ms non-zero watchdog for every device. *)
  i_watchdog_tick := FALSE;
  i_watchdog_scan_count := i_watchdog_scan_count + 1;
  IF i_watchdog_scan_count >= 10 THEN
    i_watchdog_scan_count := 0;
    i_watchdog_tick := TRUE;
    IF condenser__holding__watchdog_counter >= 65535 THEN
      condenser__holding__watchdog_counter := 1;
    ELSE
      condenser__holding__watchdog_counter := condenser__holding__watchdog_counter + 1;
    END_IF;
    IF condensate_pump__holding__watchdog_counter >= 65535 THEN
      condensate_pump__holding__watchdog_counter := 1;
    ELSE
      condensate_pump__holding__watchdog_counter := condensate_pump__holding__watchdog_counter + 1;
    END_IF;
    IF feedwater_tank__holding__watchdog_counter >= 65535 THEN
      feedwater_tank__holding__watchdog_counter := 1;
    ELSE
      feedwater_tank__holding__watchdog_counter := feedwater_tank__holding__watchdog_counter + 1;
    END_IF;
    IF feedwater_pump__holding__watchdog_counter >= 65535 THEN
      feedwater_pump__holding__watchdog_counter := 1;
    ELSE
      feedwater_pump__holding__watchdog_counter := feedwater_pump__holding__watchdog_counter + 1;
    END_IF;
    IF boiler__holding__watchdog_counter >= 65535 THEN
      boiler__holding__watchdog_counter := 1;
    ELSE
      boiler__holding__watchdog_counter := boiler__holding__watchdog_counter + 1;
    END_IF;
    IF steam_valve__holding__watchdog_counter >= 65535 THEN
      steam_valve__holding__watchdog_counter := 1;
    ELSE
      steam_valve__holding__watchdog_counter := steam_valve__holding__watchdog_counter + 1;
    END_IF;
    IF turbine__holding__watchdog_counter >= 65535 THEN
      turbine__holding__watchdog_counter := 1;
    ELSE
      turbine__holding__watchdog_counter := turbine__holding__watchdog_counter + 1;
    END_IF;
    IF generator__holding__watchdog_counter >= 65535 THEN
      generator__holding__watchdog_counter := 1;
    ELSE
      generator__holding__watchdog_counter := generator__holding__watchdog_counter + 1;
    END_IF;
  END_IF;

  (* Echo lags the counter because FC4 polls every 250 ms; an unchanged
     mismatch for 15 ticks is a communication failure. *)
  IF i_watchdog_tick THEN
    IF (condenser__input__watchdog_echo = condenser__holding__watchdog_counter) OR (condenser__input__watchdog_echo <> i_condenser_last_echo) THEN
      i_condenser_last_echo := condenser__input__watchdog_echo;
      i_condenser_echo_stale_ticks := 0;
    ELSE
      IF i_condenser_echo_stale_ticks < 65535 THEN
        i_condenser_echo_stale_ticks := i_condenser_echo_stale_ticks + 1;
      END_IF;
    END_IF;
    i_condenser_comm_lost := i_condenser_echo_stale_ticks >= 15;
    IF (condensate_pump__input__watchdog_echo = condensate_pump__holding__watchdog_counter) OR (condensate_pump__input__watchdog_echo <> i_condensate_pump_last_echo) THEN
      i_condensate_pump_last_echo := condensate_pump__input__watchdog_echo;
      i_condensate_pump_echo_stale_ticks := 0;
    ELSE
      IF i_condensate_pump_echo_stale_ticks < 65535 THEN
        i_condensate_pump_echo_stale_ticks := i_condensate_pump_echo_stale_ticks + 1;
      END_IF;
    END_IF;
    i_condensate_pump_comm_lost := i_condensate_pump_echo_stale_ticks >= 15;
    IF (feedwater_tank__input__watchdog_echo = feedwater_tank__holding__watchdog_counter) OR (feedwater_tank__input__watchdog_echo <> i_feedwater_tank_last_echo) THEN
      i_feedwater_tank_last_echo := feedwater_tank__input__watchdog_echo;
      i_feedwater_tank_echo_stale_ticks := 0;
    ELSE
      IF i_feedwater_tank_echo_stale_ticks < 65535 THEN
        i_feedwater_tank_echo_stale_ticks := i_feedwater_tank_echo_stale_ticks + 1;
      END_IF;
    END_IF;
    i_feedwater_tank_comm_lost := i_feedwater_tank_echo_stale_ticks >= 15;
    IF (feedwater_pump__input__watchdog_echo = feedwater_pump__holding__watchdog_counter) OR (feedwater_pump__input__watchdog_echo <> i_feedwater_pump_last_echo) THEN
      i_feedwater_pump_last_echo := feedwater_pump__input__watchdog_echo;
      i_feedwater_pump_echo_stale_ticks := 0;
    ELSE
      IF i_feedwater_pump_echo_stale_ticks < 65535 THEN
        i_feedwater_pump_echo_stale_ticks := i_feedwater_pump_echo_stale_ticks + 1;
      END_IF;
    END_IF;
    i_feedwater_pump_comm_lost := i_feedwater_pump_echo_stale_ticks >= 15;
    IF (boiler__input__watchdog_echo = boiler__holding__watchdog_counter) OR (boiler__input__watchdog_echo <> i_boiler_last_echo) THEN
      i_boiler_last_echo := boiler__input__watchdog_echo;
      i_boiler_echo_stale_ticks := 0;
    ELSE
      IF i_boiler_echo_stale_ticks < 65535 THEN
        i_boiler_echo_stale_ticks := i_boiler_echo_stale_ticks + 1;
      END_IF;
    END_IF;
    i_boiler_comm_lost := i_boiler_echo_stale_ticks >= 15;
    IF (steam_valve__input__watchdog_echo = steam_valve__holding__watchdog_counter) OR (steam_valve__input__watchdog_echo <> i_steam_valve_last_echo) THEN
      i_steam_valve_last_echo := steam_valve__input__watchdog_echo;
      i_steam_valve_echo_stale_ticks := 0;
    ELSE
      IF i_steam_valve_echo_stale_ticks < 65535 THEN
        i_steam_valve_echo_stale_ticks := i_steam_valve_echo_stale_ticks + 1;
      END_IF;
    END_IF;
    i_steam_valve_comm_lost := i_steam_valve_echo_stale_ticks >= 15;
    IF (turbine__input__watchdog_echo = turbine__holding__watchdog_counter) OR (turbine__input__watchdog_echo <> i_turbine_last_echo) THEN
      i_turbine_last_echo := turbine__input__watchdog_echo;
      i_turbine_echo_stale_ticks := 0;
    ELSE
      IF i_turbine_echo_stale_ticks < 65535 THEN
        i_turbine_echo_stale_ticks := i_turbine_echo_stale_ticks + 1;
      END_IF;
    END_IF;
    i_turbine_comm_lost := i_turbine_echo_stale_ticks >= 15;
    IF (generator__input__watchdog_echo = generator__holding__watchdog_counter) OR (generator__input__watchdog_echo <> i_generator_last_echo) THEN
      i_generator_last_echo := generator__input__watchdog_echo;
      i_generator_echo_stale_ticks := 0;
    ELSE
      IF i_generator_echo_stale_ticks < 65535 THEN
        i_generator_echo_stale_ticks := i_generator_echo_stale_ticks + 1;
      END_IF;
    END_IF;
    i_generator_comm_lost := i_generator_echo_stale_ticks >= 15;
  END_IF;

  (* Communication loss is a status, not an action: the devices keep
     running on their own regulators. *)
  i_plant_comm_lost := i_condenser_comm_lost OR i_condensate_pump_comm_lost OR i_feedwater_tank_comm_lost OR i_feedwater_pump_comm_lost OR i_boiler_comm_lost OR i_steam_valve_comm_lost OR i_turbine_comm_lost OR i_generator_comm_lost;

  (* Pulse commands are stretched to about 160 ms
     then cleared.  EMERGENCY_STOP and FORCE_SAFE are maintained. *)
  IF condenser__coil__start AND NOT i_condenser_start_active THEN
    i_condenser_start_active := TRUE;
    i_condenser_start_scans := 0;
  END_IF;
  IF i_condenser_start_active THEN
    i_condenser_start_scans := i_condenser_start_scans + 1;
    IF i_condenser_start_scans >= 8 THEN
      condenser__coil__start := FALSE;
      i_condenser_start_active := FALSE;
      i_condenser_start_scans := 0;
    END_IF;
  END_IF;
  IF condenser__coil__stop AND NOT i_condenser_stop_active THEN
    i_condenser_stop_active := TRUE;
    i_condenser_stop_scans := 0;
  END_IF;
  IF i_condenser_stop_active THEN
    i_condenser_stop_scans := i_condenser_stop_scans + 1;
    IF i_condenser_stop_scans >= 8 THEN
      condenser__coil__stop := FALSE;
      i_condenser_stop_active := FALSE;
      i_condenser_stop_scans := 0;
    END_IF;
  END_IF;
  IF condenser__coil__reset_trip AND NOT i_condenser_reset_trip_active THEN
    i_condenser_reset_trip_active := TRUE;
    i_condenser_reset_trip_scans := 0;
    IF condenser__holding__command_sequence >= 65535 THEN
      condenser__holding__command_sequence := 1;
    ELSE
      condenser__holding__command_sequence := condenser__holding__command_sequence + 1;
    END_IF;
    condenser__holding__reset_key := 42330;
  END_IF;
  IF i_condenser_reset_trip_active THEN
    i_condenser_reset_trip_scans := i_condenser_reset_trip_scans + 1;
    IF i_condenser_reset_trip_scans >= 8 THEN
      condenser__coil__reset_trip := FALSE;
      i_condenser_reset_trip_active := FALSE;
      i_condenser_reset_trip_scans := 0;
      condenser__holding__reset_key := 0;
    END_IF;
  END_IF;
  IF condenser__coil__ack_alarm AND NOT i_condenser_ack_alarm_active THEN
    i_condenser_ack_alarm_active := TRUE;
    i_condenser_ack_alarm_scans := 0;
  END_IF;
  IF i_condenser_ack_alarm_active THEN
    i_condenser_ack_alarm_scans := i_condenser_ack_alarm_scans + 1;
    IF i_condenser_ack_alarm_scans >= 8 THEN
      condenser__coil__ack_alarm := FALSE;
      i_condenser_ack_alarm_active := FALSE;
      i_condenser_ack_alarm_scans := 0;
    END_IF;
  END_IF;
  IF condenser__coil__trip_test AND NOT i_condenser_trip_test_active THEN
    i_condenser_trip_test_active := TRUE;
    i_condenser_trip_test_scans := 0;
  END_IF;
  IF i_condenser_trip_test_active THEN
    i_condenser_trip_test_scans := i_condenser_trip_test_scans + 1;
    IF i_condenser_trip_test_scans >= 8 THEN
      condenser__coil__trip_test := FALSE;
      i_condenser_trip_test_active := FALSE;
      i_condenser_trip_test_scans := 0;
    END_IF;
  END_IF;
  IF condenser__coil__clear_totalizer AND NOT i_condenser_clear_totalizer_active THEN
    i_condenser_clear_totalizer_active := TRUE;
    i_condenser_clear_totalizer_scans := 0;
  END_IF;
  IF i_condenser_clear_totalizer_active THEN
    i_condenser_clear_totalizer_scans := i_condenser_clear_totalizer_scans + 1;
    IF i_condenser_clear_totalizer_scans >= 8 THEN
      condenser__coil__clear_totalizer := FALSE;
      i_condenser_clear_totalizer_active := FALSE;
      i_condenser_clear_totalizer_scans := 0;
    END_IF;
  END_IF;
  IF condensate_pump__coil__start AND NOT i_condensate_pump_start_active THEN
    i_condensate_pump_start_active := TRUE;
    i_condensate_pump_start_scans := 0;
  END_IF;
  IF i_condensate_pump_start_active THEN
    i_condensate_pump_start_scans := i_condensate_pump_start_scans + 1;
    IF i_condensate_pump_start_scans >= 8 THEN
      condensate_pump__coil__start := FALSE;
      i_condensate_pump_start_active := FALSE;
      i_condensate_pump_start_scans := 0;
    END_IF;
  END_IF;
  IF condensate_pump__coil__stop AND NOT i_condensate_pump_stop_active THEN
    i_condensate_pump_stop_active := TRUE;
    i_condensate_pump_stop_scans := 0;
  END_IF;
  IF i_condensate_pump_stop_active THEN
    i_condensate_pump_stop_scans := i_condensate_pump_stop_scans + 1;
    IF i_condensate_pump_stop_scans >= 8 THEN
      condensate_pump__coil__stop := FALSE;
      i_condensate_pump_stop_active := FALSE;
      i_condensate_pump_stop_scans := 0;
    END_IF;
  END_IF;
  IF condensate_pump__coil__reset_trip AND NOT i_condensate_pump_reset_trip_active THEN
    i_condensate_pump_reset_trip_active := TRUE;
    i_condensate_pump_reset_trip_scans := 0;
    IF condensate_pump__holding__command_sequence >= 65535 THEN
      condensate_pump__holding__command_sequence := 1;
    ELSE
      condensate_pump__holding__command_sequence := condensate_pump__holding__command_sequence + 1;
    END_IF;
    condensate_pump__holding__reset_key := 42330;
  END_IF;
  IF i_condensate_pump_reset_trip_active THEN
    i_condensate_pump_reset_trip_scans := i_condensate_pump_reset_trip_scans + 1;
    IF i_condensate_pump_reset_trip_scans >= 8 THEN
      condensate_pump__coil__reset_trip := FALSE;
      i_condensate_pump_reset_trip_active := FALSE;
      i_condensate_pump_reset_trip_scans := 0;
      condensate_pump__holding__reset_key := 0;
    END_IF;
  END_IF;
  IF condensate_pump__coil__ack_alarm AND NOT i_condensate_pump_ack_alarm_active THEN
    i_condensate_pump_ack_alarm_active := TRUE;
    i_condensate_pump_ack_alarm_scans := 0;
  END_IF;
  IF i_condensate_pump_ack_alarm_active THEN
    i_condensate_pump_ack_alarm_scans := i_condensate_pump_ack_alarm_scans + 1;
    IF i_condensate_pump_ack_alarm_scans >= 8 THEN
      condensate_pump__coil__ack_alarm := FALSE;
      i_condensate_pump_ack_alarm_active := FALSE;
      i_condensate_pump_ack_alarm_scans := 0;
    END_IF;
  END_IF;
  IF condensate_pump__coil__trip_test AND NOT i_condensate_pump_trip_test_active THEN
    i_condensate_pump_trip_test_active := TRUE;
    i_condensate_pump_trip_test_scans := 0;
  END_IF;
  IF i_condensate_pump_trip_test_active THEN
    i_condensate_pump_trip_test_scans := i_condensate_pump_trip_test_scans + 1;
    IF i_condensate_pump_trip_test_scans >= 8 THEN
      condensate_pump__coil__trip_test := FALSE;
      i_condensate_pump_trip_test_active := FALSE;
      i_condensate_pump_trip_test_scans := 0;
    END_IF;
  END_IF;
  IF condensate_pump__coil__clear_totalizer AND NOT i_condensate_pump_clear_totalizer_active THEN
    i_condensate_pump_clear_totalizer_active := TRUE;
    i_condensate_pump_clear_totalizer_scans := 0;
  END_IF;
  IF i_condensate_pump_clear_totalizer_active THEN
    i_condensate_pump_clear_totalizer_scans := i_condensate_pump_clear_totalizer_scans + 1;
    IF i_condensate_pump_clear_totalizer_scans >= 8 THEN
      condensate_pump__coil__clear_totalizer := FALSE;
      i_condensate_pump_clear_totalizer_active := FALSE;
      i_condensate_pump_clear_totalizer_scans := 0;
    END_IF;
  END_IF;
  IF feedwater_tank__coil__start AND NOT i_feedwater_tank_start_active THEN
    i_feedwater_tank_start_active := TRUE;
    i_feedwater_tank_start_scans := 0;
  END_IF;
  IF i_feedwater_tank_start_active THEN
    i_feedwater_tank_start_scans := i_feedwater_tank_start_scans + 1;
    IF i_feedwater_tank_start_scans >= 8 THEN
      feedwater_tank__coil__start := FALSE;
      i_feedwater_tank_start_active := FALSE;
      i_feedwater_tank_start_scans := 0;
    END_IF;
  END_IF;
  IF feedwater_tank__coil__stop AND NOT i_feedwater_tank_stop_active THEN
    i_feedwater_tank_stop_active := TRUE;
    i_feedwater_tank_stop_scans := 0;
  END_IF;
  IF i_feedwater_tank_stop_active THEN
    i_feedwater_tank_stop_scans := i_feedwater_tank_stop_scans + 1;
    IF i_feedwater_tank_stop_scans >= 8 THEN
      feedwater_tank__coil__stop := FALSE;
      i_feedwater_tank_stop_active := FALSE;
      i_feedwater_tank_stop_scans := 0;
    END_IF;
  END_IF;
  IF feedwater_tank__coil__reset_trip AND NOT i_feedwater_tank_reset_trip_active THEN
    i_feedwater_tank_reset_trip_active := TRUE;
    i_feedwater_tank_reset_trip_scans := 0;
    IF feedwater_tank__holding__command_sequence >= 65535 THEN
      feedwater_tank__holding__command_sequence := 1;
    ELSE
      feedwater_tank__holding__command_sequence := feedwater_tank__holding__command_sequence + 1;
    END_IF;
    feedwater_tank__holding__reset_key := 42330;
  END_IF;
  IF i_feedwater_tank_reset_trip_active THEN
    i_feedwater_tank_reset_trip_scans := i_feedwater_tank_reset_trip_scans + 1;
    IF i_feedwater_tank_reset_trip_scans >= 8 THEN
      feedwater_tank__coil__reset_trip := FALSE;
      i_feedwater_tank_reset_trip_active := FALSE;
      i_feedwater_tank_reset_trip_scans := 0;
      feedwater_tank__holding__reset_key := 0;
    END_IF;
  END_IF;
  IF feedwater_tank__coil__ack_alarm AND NOT i_feedwater_tank_ack_alarm_active THEN
    i_feedwater_tank_ack_alarm_active := TRUE;
    i_feedwater_tank_ack_alarm_scans := 0;
  END_IF;
  IF i_feedwater_tank_ack_alarm_active THEN
    i_feedwater_tank_ack_alarm_scans := i_feedwater_tank_ack_alarm_scans + 1;
    IF i_feedwater_tank_ack_alarm_scans >= 8 THEN
      feedwater_tank__coil__ack_alarm := FALSE;
      i_feedwater_tank_ack_alarm_active := FALSE;
      i_feedwater_tank_ack_alarm_scans := 0;
    END_IF;
  END_IF;
  IF feedwater_tank__coil__trip_test AND NOT i_feedwater_tank_trip_test_active THEN
    i_feedwater_tank_trip_test_active := TRUE;
    i_feedwater_tank_trip_test_scans := 0;
  END_IF;
  IF i_feedwater_tank_trip_test_active THEN
    i_feedwater_tank_trip_test_scans := i_feedwater_tank_trip_test_scans + 1;
    IF i_feedwater_tank_trip_test_scans >= 8 THEN
      feedwater_tank__coil__trip_test := FALSE;
      i_feedwater_tank_trip_test_active := FALSE;
      i_feedwater_tank_trip_test_scans := 0;
    END_IF;
  END_IF;
  IF feedwater_tank__coil__clear_totalizer AND NOT i_feedwater_tank_clear_totalizer_active THEN
    i_feedwater_tank_clear_totalizer_active := TRUE;
    i_feedwater_tank_clear_totalizer_scans := 0;
  END_IF;
  IF i_feedwater_tank_clear_totalizer_active THEN
    i_feedwater_tank_clear_totalizer_scans := i_feedwater_tank_clear_totalizer_scans + 1;
    IF i_feedwater_tank_clear_totalizer_scans >= 8 THEN
      feedwater_tank__coil__clear_totalizer := FALSE;
      i_feedwater_tank_clear_totalizer_active := FALSE;
      i_feedwater_tank_clear_totalizer_scans := 0;
    END_IF;
  END_IF;
  IF feedwater_pump__coil__start AND NOT i_feedwater_pump_start_active THEN
    i_feedwater_pump_start_active := TRUE;
    i_feedwater_pump_start_scans := 0;
  END_IF;
  IF i_feedwater_pump_start_active THEN
    i_feedwater_pump_start_scans := i_feedwater_pump_start_scans + 1;
    IF i_feedwater_pump_start_scans >= 8 THEN
      feedwater_pump__coil__start := FALSE;
      i_feedwater_pump_start_active := FALSE;
      i_feedwater_pump_start_scans := 0;
    END_IF;
  END_IF;
  IF feedwater_pump__coil__stop AND NOT i_feedwater_pump_stop_active THEN
    i_feedwater_pump_stop_active := TRUE;
    i_feedwater_pump_stop_scans := 0;
  END_IF;
  IF i_feedwater_pump_stop_active THEN
    i_feedwater_pump_stop_scans := i_feedwater_pump_stop_scans + 1;
    IF i_feedwater_pump_stop_scans >= 8 THEN
      feedwater_pump__coil__stop := FALSE;
      i_feedwater_pump_stop_active := FALSE;
      i_feedwater_pump_stop_scans := 0;
    END_IF;
  END_IF;
  IF feedwater_pump__coil__reset_trip AND NOT i_feedwater_pump_reset_trip_active THEN
    i_feedwater_pump_reset_trip_active := TRUE;
    i_feedwater_pump_reset_trip_scans := 0;
    IF feedwater_pump__holding__command_sequence >= 65535 THEN
      feedwater_pump__holding__command_sequence := 1;
    ELSE
      feedwater_pump__holding__command_sequence := feedwater_pump__holding__command_sequence + 1;
    END_IF;
    feedwater_pump__holding__reset_key := 42330;
  END_IF;
  IF i_feedwater_pump_reset_trip_active THEN
    i_feedwater_pump_reset_trip_scans := i_feedwater_pump_reset_trip_scans + 1;
    IF i_feedwater_pump_reset_trip_scans >= 8 THEN
      feedwater_pump__coil__reset_trip := FALSE;
      i_feedwater_pump_reset_trip_active := FALSE;
      i_feedwater_pump_reset_trip_scans := 0;
      feedwater_pump__holding__reset_key := 0;
    END_IF;
  END_IF;
  IF feedwater_pump__coil__ack_alarm AND NOT i_feedwater_pump_ack_alarm_active THEN
    i_feedwater_pump_ack_alarm_active := TRUE;
    i_feedwater_pump_ack_alarm_scans := 0;
  END_IF;
  IF i_feedwater_pump_ack_alarm_active THEN
    i_feedwater_pump_ack_alarm_scans := i_feedwater_pump_ack_alarm_scans + 1;
    IF i_feedwater_pump_ack_alarm_scans >= 8 THEN
      feedwater_pump__coil__ack_alarm := FALSE;
      i_feedwater_pump_ack_alarm_active := FALSE;
      i_feedwater_pump_ack_alarm_scans := 0;
    END_IF;
  END_IF;
  IF feedwater_pump__coil__trip_test AND NOT i_feedwater_pump_trip_test_active THEN
    i_feedwater_pump_trip_test_active := TRUE;
    i_feedwater_pump_trip_test_scans := 0;
  END_IF;
  IF i_feedwater_pump_trip_test_active THEN
    i_feedwater_pump_trip_test_scans := i_feedwater_pump_trip_test_scans + 1;
    IF i_feedwater_pump_trip_test_scans >= 8 THEN
      feedwater_pump__coil__trip_test := FALSE;
      i_feedwater_pump_trip_test_active := FALSE;
      i_feedwater_pump_trip_test_scans := 0;
    END_IF;
  END_IF;
  IF feedwater_pump__coil__clear_totalizer AND NOT i_feedwater_pump_clear_totalizer_active THEN
    i_feedwater_pump_clear_totalizer_active := TRUE;
    i_feedwater_pump_clear_totalizer_scans := 0;
  END_IF;
  IF i_feedwater_pump_clear_totalizer_active THEN
    i_feedwater_pump_clear_totalizer_scans := i_feedwater_pump_clear_totalizer_scans + 1;
    IF i_feedwater_pump_clear_totalizer_scans >= 8 THEN
      feedwater_pump__coil__clear_totalizer := FALSE;
      i_feedwater_pump_clear_totalizer_active := FALSE;
      i_feedwater_pump_clear_totalizer_scans := 0;
    END_IF;
  END_IF;
  IF boiler__coil__start AND NOT i_boiler_start_active THEN
    i_boiler_start_active := TRUE;
    i_boiler_start_scans := 0;
  END_IF;
  IF i_boiler_start_active THEN
    i_boiler_start_scans := i_boiler_start_scans + 1;
    IF i_boiler_start_scans >= 8 THEN
      boiler__coil__start := FALSE;
      i_boiler_start_active := FALSE;
      i_boiler_start_scans := 0;
    END_IF;
  END_IF;
  IF boiler__coil__stop AND NOT i_boiler_stop_active THEN
    i_boiler_stop_active := TRUE;
    i_boiler_stop_scans := 0;
  END_IF;
  IF i_boiler_stop_active THEN
    i_boiler_stop_scans := i_boiler_stop_scans + 1;
    IF i_boiler_stop_scans >= 8 THEN
      boiler__coil__stop := FALSE;
      i_boiler_stop_active := FALSE;
      i_boiler_stop_scans := 0;
    END_IF;
  END_IF;
  IF boiler__coil__reset_trip AND NOT i_boiler_reset_trip_active THEN
    i_boiler_reset_trip_active := TRUE;
    i_boiler_reset_trip_scans := 0;
    IF boiler__holding__command_sequence >= 65535 THEN
      boiler__holding__command_sequence := 1;
    ELSE
      boiler__holding__command_sequence := boiler__holding__command_sequence + 1;
    END_IF;
    boiler__holding__reset_key := 42330;
  END_IF;
  IF i_boiler_reset_trip_active THEN
    i_boiler_reset_trip_scans := i_boiler_reset_trip_scans + 1;
    IF i_boiler_reset_trip_scans >= 8 THEN
      boiler__coil__reset_trip := FALSE;
      i_boiler_reset_trip_active := FALSE;
      i_boiler_reset_trip_scans := 0;
      boiler__holding__reset_key := 0;
    END_IF;
  END_IF;
  IF boiler__coil__ack_alarm AND NOT i_boiler_ack_alarm_active THEN
    i_boiler_ack_alarm_active := TRUE;
    i_boiler_ack_alarm_scans := 0;
  END_IF;
  IF i_boiler_ack_alarm_active THEN
    i_boiler_ack_alarm_scans := i_boiler_ack_alarm_scans + 1;
    IF i_boiler_ack_alarm_scans >= 8 THEN
      boiler__coil__ack_alarm := FALSE;
      i_boiler_ack_alarm_active := FALSE;
      i_boiler_ack_alarm_scans := 0;
    END_IF;
  END_IF;
  IF boiler__coil__trip_test AND NOT i_boiler_trip_test_active THEN
    i_boiler_trip_test_active := TRUE;
    i_boiler_trip_test_scans := 0;
  END_IF;
  IF i_boiler_trip_test_active THEN
    i_boiler_trip_test_scans := i_boiler_trip_test_scans + 1;
    IF i_boiler_trip_test_scans >= 8 THEN
      boiler__coil__trip_test := FALSE;
      i_boiler_trip_test_active := FALSE;
      i_boiler_trip_test_scans := 0;
    END_IF;
  END_IF;
  IF boiler__coil__clear_totalizer AND NOT i_boiler_clear_totalizer_active THEN
    i_boiler_clear_totalizer_active := TRUE;
    i_boiler_clear_totalizer_scans := 0;
  END_IF;
  IF i_boiler_clear_totalizer_active THEN
    i_boiler_clear_totalizer_scans := i_boiler_clear_totalizer_scans + 1;
    IF i_boiler_clear_totalizer_scans >= 8 THEN
      boiler__coil__clear_totalizer := FALSE;
      i_boiler_clear_totalizer_active := FALSE;
      i_boiler_clear_totalizer_scans := 0;
    END_IF;
  END_IF;
  IF steam_valve__coil__start AND NOT i_steam_valve_start_active THEN
    i_steam_valve_start_active := TRUE;
    i_steam_valve_start_scans := 0;
  END_IF;
  IF i_steam_valve_start_active THEN
    i_steam_valve_start_scans := i_steam_valve_start_scans + 1;
    IF i_steam_valve_start_scans >= 8 THEN
      steam_valve__coil__start := FALSE;
      i_steam_valve_start_active := FALSE;
      i_steam_valve_start_scans := 0;
    END_IF;
  END_IF;
  IF steam_valve__coil__stop AND NOT i_steam_valve_stop_active THEN
    i_steam_valve_stop_active := TRUE;
    i_steam_valve_stop_scans := 0;
  END_IF;
  IF i_steam_valve_stop_active THEN
    i_steam_valve_stop_scans := i_steam_valve_stop_scans + 1;
    IF i_steam_valve_stop_scans >= 8 THEN
      steam_valve__coil__stop := FALSE;
      i_steam_valve_stop_active := FALSE;
      i_steam_valve_stop_scans := 0;
    END_IF;
  END_IF;
  IF steam_valve__coil__reset_trip AND NOT i_steam_valve_reset_trip_active THEN
    i_steam_valve_reset_trip_active := TRUE;
    i_steam_valve_reset_trip_scans := 0;
    IF steam_valve__holding__command_sequence >= 65535 THEN
      steam_valve__holding__command_sequence := 1;
    ELSE
      steam_valve__holding__command_sequence := steam_valve__holding__command_sequence + 1;
    END_IF;
    steam_valve__holding__reset_key := 42330;
  END_IF;
  IF i_steam_valve_reset_trip_active THEN
    i_steam_valve_reset_trip_scans := i_steam_valve_reset_trip_scans + 1;
    IF i_steam_valve_reset_trip_scans >= 8 THEN
      steam_valve__coil__reset_trip := FALSE;
      i_steam_valve_reset_trip_active := FALSE;
      i_steam_valve_reset_trip_scans := 0;
      steam_valve__holding__reset_key := 0;
    END_IF;
  END_IF;
  IF steam_valve__coil__ack_alarm AND NOT i_steam_valve_ack_alarm_active THEN
    i_steam_valve_ack_alarm_active := TRUE;
    i_steam_valve_ack_alarm_scans := 0;
  END_IF;
  IF i_steam_valve_ack_alarm_active THEN
    i_steam_valve_ack_alarm_scans := i_steam_valve_ack_alarm_scans + 1;
    IF i_steam_valve_ack_alarm_scans >= 8 THEN
      steam_valve__coil__ack_alarm := FALSE;
      i_steam_valve_ack_alarm_active := FALSE;
      i_steam_valve_ack_alarm_scans := 0;
    END_IF;
  END_IF;
  IF steam_valve__coil__trip_test AND NOT i_steam_valve_trip_test_active THEN
    i_steam_valve_trip_test_active := TRUE;
    i_steam_valve_trip_test_scans := 0;
  END_IF;
  IF i_steam_valve_trip_test_active THEN
    i_steam_valve_trip_test_scans := i_steam_valve_trip_test_scans + 1;
    IF i_steam_valve_trip_test_scans >= 8 THEN
      steam_valve__coil__trip_test := FALSE;
      i_steam_valve_trip_test_active := FALSE;
      i_steam_valve_trip_test_scans := 0;
    END_IF;
  END_IF;
  IF steam_valve__coil__clear_totalizer AND NOT i_steam_valve_clear_totalizer_active THEN
    i_steam_valve_clear_totalizer_active := TRUE;
    i_steam_valve_clear_totalizer_scans := 0;
  END_IF;
  IF i_steam_valve_clear_totalizer_active THEN
    i_steam_valve_clear_totalizer_scans := i_steam_valve_clear_totalizer_scans + 1;
    IF i_steam_valve_clear_totalizer_scans >= 8 THEN
      steam_valve__coil__clear_totalizer := FALSE;
      i_steam_valve_clear_totalizer_active := FALSE;
      i_steam_valve_clear_totalizer_scans := 0;
    END_IF;
  END_IF;
  IF turbine__coil__start AND NOT i_turbine_start_active THEN
    i_turbine_start_active := TRUE;
    i_turbine_start_scans := 0;
  END_IF;
  IF i_turbine_start_active THEN
    i_turbine_start_scans := i_turbine_start_scans + 1;
    IF i_turbine_start_scans >= 8 THEN
      turbine__coil__start := FALSE;
      i_turbine_start_active := FALSE;
      i_turbine_start_scans := 0;
    END_IF;
  END_IF;
  IF turbine__coil__stop AND NOT i_turbine_stop_active THEN
    i_turbine_stop_active := TRUE;
    i_turbine_stop_scans := 0;
  END_IF;
  IF i_turbine_stop_active THEN
    i_turbine_stop_scans := i_turbine_stop_scans + 1;
    IF i_turbine_stop_scans >= 8 THEN
      turbine__coil__stop := FALSE;
      i_turbine_stop_active := FALSE;
      i_turbine_stop_scans := 0;
    END_IF;
  END_IF;
  IF turbine__coil__reset_trip AND NOT i_turbine_reset_trip_active THEN
    i_turbine_reset_trip_active := TRUE;
    i_turbine_reset_trip_scans := 0;
    IF turbine__holding__command_sequence >= 65535 THEN
      turbine__holding__command_sequence := 1;
    ELSE
      turbine__holding__command_sequence := turbine__holding__command_sequence + 1;
    END_IF;
    turbine__holding__reset_key := 42330;
  END_IF;
  IF i_turbine_reset_trip_active THEN
    i_turbine_reset_trip_scans := i_turbine_reset_trip_scans + 1;
    IF i_turbine_reset_trip_scans >= 8 THEN
      turbine__coil__reset_trip := FALSE;
      i_turbine_reset_trip_active := FALSE;
      i_turbine_reset_trip_scans := 0;
      turbine__holding__reset_key := 0;
    END_IF;
  END_IF;
  IF turbine__coil__ack_alarm AND NOT i_turbine_ack_alarm_active THEN
    i_turbine_ack_alarm_active := TRUE;
    i_turbine_ack_alarm_scans := 0;
  END_IF;
  IF i_turbine_ack_alarm_active THEN
    i_turbine_ack_alarm_scans := i_turbine_ack_alarm_scans + 1;
    IF i_turbine_ack_alarm_scans >= 8 THEN
      turbine__coil__ack_alarm := FALSE;
      i_turbine_ack_alarm_active := FALSE;
      i_turbine_ack_alarm_scans := 0;
    END_IF;
  END_IF;
  IF turbine__coil__trip_test AND NOT i_turbine_trip_test_active THEN
    i_turbine_trip_test_active := TRUE;
    i_turbine_trip_test_scans := 0;
  END_IF;
  IF i_turbine_trip_test_active THEN
    i_turbine_trip_test_scans := i_turbine_trip_test_scans + 1;
    IF i_turbine_trip_test_scans >= 8 THEN
      turbine__coil__trip_test := FALSE;
      i_turbine_trip_test_active := FALSE;
      i_turbine_trip_test_scans := 0;
    END_IF;
  END_IF;
  IF turbine__coil__clear_totalizer AND NOT i_turbine_clear_totalizer_active THEN
    i_turbine_clear_totalizer_active := TRUE;
    i_turbine_clear_totalizer_scans := 0;
  END_IF;
  IF i_turbine_clear_totalizer_active THEN
    i_turbine_clear_totalizer_scans := i_turbine_clear_totalizer_scans + 1;
    IF i_turbine_clear_totalizer_scans >= 8 THEN
      turbine__coil__clear_totalizer := FALSE;
      i_turbine_clear_totalizer_active := FALSE;
      i_turbine_clear_totalizer_scans := 0;
    END_IF;
  END_IF;
  IF generator__coil__start AND NOT i_generator_start_active THEN
    i_generator_start_active := TRUE;
    i_generator_start_scans := 0;
  END_IF;
  IF i_generator_start_active THEN
    i_generator_start_scans := i_generator_start_scans + 1;
    IF i_generator_start_scans >= 8 THEN
      generator__coil__start := FALSE;
      i_generator_start_active := FALSE;
      i_generator_start_scans := 0;
    END_IF;
  END_IF;
  IF generator__coil__stop AND NOT i_generator_stop_active THEN
    i_generator_stop_active := TRUE;
    i_generator_stop_scans := 0;
  END_IF;
  IF i_generator_stop_active THEN
    i_generator_stop_scans := i_generator_stop_scans + 1;
    IF i_generator_stop_scans >= 8 THEN
      generator__coil__stop := FALSE;
      i_generator_stop_active := FALSE;
      i_generator_stop_scans := 0;
    END_IF;
  END_IF;
  IF generator__coil__reset_trip AND NOT i_generator_reset_trip_active THEN
    i_generator_reset_trip_active := TRUE;
    i_generator_reset_trip_scans := 0;
    IF generator__holding__command_sequence >= 65535 THEN
      generator__holding__command_sequence := 1;
    ELSE
      generator__holding__command_sequence := generator__holding__command_sequence + 1;
    END_IF;
    generator__holding__reset_key := 42330;
  END_IF;
  IF i_generator_reset_trip_active THEN
    i_generator_reset_trip_scans := i_generator_reset_trip_scans + 1;
    IF i_generator_reset_trip_scans >= 8 THEN
      generator__coil__reset_trip := FALSE;
      i_generator_reset_trip_active := FALSE;
      i_generator_reset_trip_scans := 0;
      generator__holding__reset_key := 0;
    END_IF;
  END_IF;
  IF generator__coil__ack_alarm AND NOT i_generator_ack_alarm_active THEN
    i_generator_ack_alarm_active := TRUE;
    i_generator_ack_alarm_scans := 0;
  END_IF;
  IF i_generator_ack_alarm_active THEN
    i_generator_ack_alarm_scans := i_generator_ack_alarm_scans + 1;
    IF i_generator_ack_alarm_scans >= 8 THEN
      generator__coil__ack_alarm := FALSE;
      i_generator_ack_alarm_active := FALSE;
      i_generator_ack_alarm_scans := 0;
    END_IF;
  END_IF;
  IF generator__coil__trip_test AND NOT i_generator_trip_test_active THEN
    i_generator_trip_test_active := TRUE;
    i_generator_trip_test_scans := 0;
  END_IF;
  IF i_generator_trip_test_active THEN
    i_generator_trip_test_scans := i_generator_trip_test_scans + 1;
    IF i_generator_trip_test_scans >= 8 THEN
      generator__coil__trip_test := FALSE;
      i_generator_trip_test_active := FALSE;
      i_generator_trip_test_scans := 0;
    END_IF;
  END_IF;
  IF generator__coil__clear_totalizer AND NOT i_generator_clear_totalizer_active THEN
    i_generator_clear_totalizer_active := TRUE;
    i_generator_clear_totalizer_scans := 0;
  END_IF;
  IF i_generator_clear_totalizer_active THEN
    i_generator_clear_totalizer_scans := i_generator_clear_totalizer_scans + 1;
    IF i_generator_clear_totalizer_scans >= 8 THEN
      generator__coil__clear_totalizer := FALSE;
      i_generator_clear_totalizer_active := FALSE;
      i_generator_clear_totalizer_scans := 0;
    END_IF;
  END_IF;

  (* Rising-edge plant trip matrix, commands only. *)
  IF turbine__discrete__tripped AND NOT i_turbine_trip_prev THEN
    steam_valve__coil__stop := TRUE;
  END_IF;
  i_turbine_trip_prev := turbine__discrete__tripped;
  IF boiler__discrete__tripped AND NOT i_boiler_trip_prev THEN
    steam_valve__coil__stop := TRUE;
  END_IF;
  i_boiler_trip_prev := boiler__discrete__tripped;
  IF condenser__discrete__tripped AND NOT i_condenser_trip_prev THEN
    (* device-level interlocks are sufficient *)
  END_IF;
  i_condenser_trip_prev := condenser__discrete__tripped;
  IF feedwater_pump__discrete__tripped AND NOT i_feedwater_pump_trip_prev THEN
    boiler__coil__stop := TRUE;
  END_IF;
  i_feedwater_pump_trip_prev := feedwater_pump__discrete__tripped;
  IF condensate_pump__discrete__tripped AND NOT i_condensate_pump_trip_prev THEN
    (* device-level interlocks are sufficient *)
  END_IF;
  i_condensate_pump_trip_prev := condensate_pump__discrete__tripped;
  IF steam_valve__discrete__tripped AND NOT i_steam_valve_trip_prev THEN
    boiler__coil__stop := TRUE;
  END_IF;
  i_steam_valve_trip_prev := steam_valve__discrete__tripped;

  (* Overspeed independently stops the main steam valve. *)
  i_overspeed := (turbine__input__speed_rpm > 3150) OR turbine__discrete__tripped;
  IF i_overspeed AND NOT i_overspeed_prev THEN
    steam_valve__coil__stop := TRUE;
  END_IF;
  i_overspeed_prev := i_overspeed;
END_PROGRAM

CONFIGURATION Config0

  RESOURCE Res0 ON PLC
    TASK task0(INTERVAL := T#20ms,PRIORITY := 0);
    PROGRAM instance0 WITH task0 : main;
  END_RESOURCE
END_CONFIGURATION
